// TIA Portal project "proyecto robot" (V15)

(* hardware
DEVICE "S7-1200 station_1"  S7-1200 Station
   slot 0: "Rack_0"  S7-1200 Rack  Rack  V1.0
   slot 1: "PLC_DERECHA"  CPU 1214C AC/DC/Rly  6ES7 214-1BG31-0XB0  V3.0
   slot 2: "AI 4x13BIT/AQ 2x14BIT_1"  6ES7 234-4HE32-0XB0  V2.0
DEVICE "S7-1200 station_2"  S7-1200 Station
   slot 0: "Rack_0"  S7-1200 Rack  Rack  V1.0
   slot 1: "PLC_IZQUIERDA"  CPU 1214C AC/DC/Rly  6ES7 214-1BG31-0XB0  V3.0
DEVICE "PC-System_1"  SIMATIC PC station
   slot 0: "Estación PC SIMATIC"  Rail  SIMATIC PC-Station  V1.0
      slot 125: "Stationmanager"  Station_Manager  V6.0.4
   slot 1: "HMI_RT_1"  WinCC RT Advanced  6AV2 104-0xxxx-xxxx  15.0.0.0
      slot 33792: "Interfaz host"  Host interface
   slot 2: "IE general_1"  IE General  IE_CP  V8.2.0
*)

// ===== PLC "PLC_DERECHA"  CPU 1214C AC/DC/Rly =====

VAR_GLOBAL   // PLC tag table "Tabla de variables estándar"
   "Clock_Byte" AT %MB1 : Byte;
   "Clock_10Hz" AT %M1.0 : Bool;
   "Clock_5Hz" AT %M1.1 : Bool;
   "Clock_2.5Hz" AT %M1.2 : Bool;
   "Clock_2Hz" AT %M1.3 : Bool;
   "Clock_1.25Hz" AT %M1.4 : Bool;
   "Clock_1Hz" AT %M1.5 : Bool;
   "Clock_0.625Hz" AT %M1.6 : Bool;
   "Clock_0.5Hz" AT %M1.7 : Bool;
   "Datos recibidos" AT %MW10 : Word;
   "Valor normalizado ultrasonidos" AT %MD50 : Real;
   "Distancia" AT %MD54 : Real;
   "Valor frecuencia cinta rueda" AT %MD58 : Real;
   "Valor normalizado frecuencia rueda" AT %MD62 : Real;
   "Normalizar frecuencia cinta chasis" AT %MD66 : Real;
   "Inicialización" AT %M12.0 : Bool;
   "marca cinta rueda" AT %M100.5 : Bool;
   "marca cilindro" AT %M100.6 : Bool;
   "Rueda en posición robot" AT %M11.1 : Bool;
   "Marca cinta chasis" AT %M100.4 : Bool;
   "Tag_4" AT %M100.7 : Bool;
   "Frecuencia cinta chasis" AT %MD70 : Real;
   "DISTANCIA HMI(1)" AT %MW200 : Int;
   "Cinta Lento" AT %MD204 : Real;
   "cinta nominal" AT %MD208 : Real;
   "HMI DISTANCIA" AT %MW1000 : Int;
   "Tag_1" AT %MD1000 : DWord;
   "Tag_2" AT %MD1200 : Real;
   "Tag_3" AT %MW500 : Word;
   "Tag_5" AT %MD500 : DInt;
   "Tag_6" AT %MD5005 : Real;
   "Tag_7" AT %MD504 : Real;
END_VAR

VAR_GLOBAL   // PLC tag table "Tabla de variables_1"
   "Error de comunicación" AT %M2.0 : Bool;
   "Marcha" AT %M10.0 : Bool;
   "Paro" AT %M10.1 : Bool;
   "Seta Emergencia" AT %M10.2 : Bool;
   "Fallo robot" AT %M10.3 : Bool;
   "jn rueda cilindro" AT %M10.4 : Bool;
   "jn fallo persona" AT %M10.5 : Bool;
   "jn cinta lento" AT %M10.6 : Bool;
   "guardamotor chasis" AT %M10.7 : Bool;
   "guardamotor rueda" AT %M11.0 : Bool;
   "Ultrasonidos" AT %IW96 : Word;
   "Variador cinta rueda" AT %QW96 : Word;
   "Variador cinta chasis" AT %QW98 : Word;
   "Motor cinta rueda" AT %Q0.0 : Bool;
   "Motor cinta chasis" AT %Q0.1 : Bool;
   "Cilindro" AT %Q0.2 : Bool;
   "Señal de fallo" AT %Q0.3 : Bool;
END_VAR

VAR_GLOBAL   // PLC tag table "HMI"
   "Seta emergencia HMI" AT %M20.0 : Bool;
   "Marcha HMI" AT %M20.1 : Bool;
   "Paro HMI" AT %M20.2 : Bool;
   "Marcha cinta chasis HMI" AT %M20.3 : Bool;
   "Paro cinta chasis HMI" AT %M20.4 : Bool;
   "Marcha cinta rueda HMI" AT %M20.5 : Bool;
   "Paro cinta rueda HMI" AT %M20.6 : Bool;
   "Control cilindro HMI" AT %M20.7 : Bool;
   "Luz marcha HMI" AT %M21.0 : Bool;
   "Luz paro HMI" AT %M21.1 : Bool;
   "Luz cinta chasis" AT %M21.2 : Bool;
   "Luz cinta rueda" AT %M21.3 : Bool;
   "Luz rueda en cinta" AT %M21.4 : Bool;
   "Luz cilindro fuera" AT %M21.5 : Bool;
   "Contador de tiempo" AT %MD300 : Time;
   "Tiempo" AT %MW202 : Word;
   "Luz seta emergencia" AT %M21.6 : Bool;
   "Luz fallo persona" AT %M21.7 : Bool;
   "Luz fallo robot" AT %M22.0 : Bool;
   "Luz guardamotor chasis" AT %M22.1 : Bool;
   "Luz guardamotor rueda" AT %M22.2 : Bool;
END_VAR

DATA_BLOCK "Guarda errores"   // DB3
{ S7_Optimized_Access := 'TRUE' }
VERSION : 0.1
   VAR
      "Seta emergencia" : DTL;
      "Fallo robot" : DTL;
      "Fallo persona" : DTL;
      "Guardamotor chasis" : DTL;
      "Guardamotor rueda" : DTL;
      "Retorno emergencia" : Int;
      "Retorno robot" : Int;
      "Retorno persona" : Int;
      "Retorno Guardamotor chasis" : Int;
      "Retorno guardamotor rueda" : Int;
   END_VAR
BEGIN
END_DATA_BLOCK

DATA_BLOCK "Velocidades"   // DB5
{ S7_Optimized_Access := 'TRUE' }
VERSION : 0.1
   VAR
      "Velocidad Lento" : Real := 10.5;
      "Velocidad Nominal" : Real := 40.0;
      "Velocidad cinta chasis" : Real := 5.0;
   END_VAR
BEGIN
END_DATA_BLOCK

// folder: System blocks/Program resources

DATA_BLOCK "PLC_DERECHA_Receive_DB"   // DB1
{ S7_Optimized_Access := 'TRUE' }
AUTHOR : SIMATIC
FAMILY : MC7Plus
NAME : TCON_Prm
VERSION : 1.0
// stored: InstanceOfName TCON_Param
"TCON_Param"
BEGIN
   ID := 1;
   REM_TSAP_ID_LEN := 0;
   LOCAL_TSAP_ID[1] := B#16#07;
   LOCAL_TSAP_ID[2] := B#16#D0;
   LOCAL_TSAP_ID_LEN := 2;
   ACTIVE_EST := false;
   REM_STADDR[1] := 172;
   REM_STADDR[2] := 26;
   REM_STADDR[3] := 20;
   REM_STADDR[4] := 50;
END_DATA_BLOCK

DATA_BLOCK "IEC_Timer_0_DB"   // DB4
{ S7_Optimized_Access := 'TRUE' }
AUTHOR : Simatic
FAMILY : IEC
NAME : IEC_TMR
VERSION : 1.0
// stored: InstanceOfName IEC_TIMER
"IEC_TIMER"
BEGIN
END_DATA_BLOCK

// folder: (top level)

FUNCTION "Cinta rueda" : Void   // FC1, LAD
{ S7_Optimized_Access := 'TRUE' }
VERSION : 0.1
   VAR_INPUT
      "Jetson Nano velocidad" : Bool;
      "Jetson Nano Rueda posición" : Bool;
      "Seta Emergencia" : Bool;
      "Fallo persona" : Bool;
      "Fallo robot" : Bool;
      Marcha : Bool;
      "Rueda abajo rampa" : Bool;
      Paro : Bool;
      "guardamotor chasis" : Bool;
      "guardamotor rueda" : Bool;
      Ultrasonidos : Real;
   END_VAR
   VAR_OUTPUT
      "Frecuencia cinta" : Int;
      "Activar cinta" : Bool;
   END_VAR
   VAR_IN_OUT
      Cilindro : Bool;
   END_VAR
BEGIN

REGION Network 1
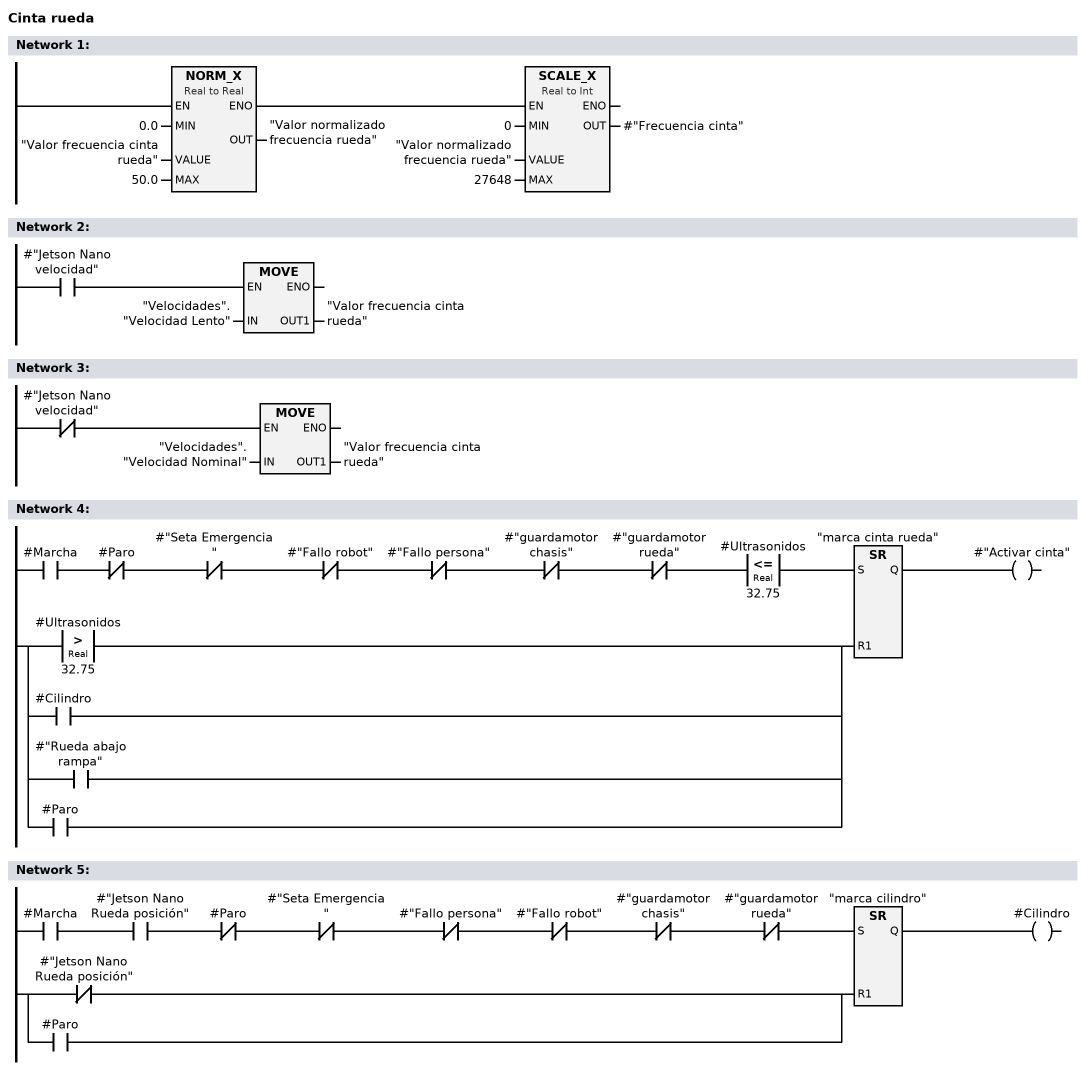
   RUNG wire#powerrail
      { S7_Templates := "[SrcType := Real, DestType := Real]"; S7_GenerateENO := "TRUE" } Normalize(min := 0.0, value := "Valor frecuencia cinta rueda", max := 50.0, out => "Valor normalizado frecuencia rueda")
      { S7_Templates := "[SrcType := Real, DestType := Int]"; S7_GenerateENO := "TRUE" } Scale(min := 0, value := "Valor normalizado frecuencia rueda", max := 27648, out => #"Frecuencia cinta")
   END_RUNG
   // the same network as SCL:
   // ENO of a box is taken as its EN; it also drops when the box reports an error
   "Valor normalizado frecuencia rueda" := NORM_X(MIN := 0.0, VALUE := "Valor frecuencia cinta rueda", MAX := 50.0);
   #"Frecuencia cinta" := SCALE_X(MIN := 0, VALUE := "Valor normalizado frecuencia rueda", MAX := 27648);
END_REGION

REGION Network 2
   RUNG wire#powerrail
      Contact( #"Jetson Nano velocidad" )
      { S7_GenerateENO := "TRUE" } Move(in := "Velocidades"."Velocidad Lento", out1 => "Valor frecuencia cinta rueda")
   END_RUNG
   // the same network as SCL:
   IF #"Jetson Nano velocidad" THEN
       "Valor frecuencia cinta rueda" := "Velocidades"."Velocidad Lento";
   END_IF;
END_REGION

REGION Network 3
   RUNG wire#powerrail
      I_Contact( #"Jetson Nano velocidad" )
      { S7_GenerateENO := "TRUE" } Move(in := "Velocidades"."Velocidad Nominal", out1 => "Valor frecuencia cinta rueda")
   END_RUNG
   // the same network as SCL:
   IF NOT #"Jetson Nano velocidad" THEN
       "Valor frecuencia cinta rueda" := "Velocidades"."Velocidad Nominal";
   END_IF;
END_REGION

REGION Network 4
   RUNG wire#powerrail
      Contact( #Marcha )
      I_Contact( #Paro )
      I_Contact( #"Seta Emergencia" )
      I_Contact( #"Fallo robot" )
      I_Contact( #"Fallo persona" )
      I_Contact( #"guardamotor chasis" )
      I_Contact( #"guardamotor rueda" )
      { S7_Templates := "SrcType := Real" } LE_Contact(in1 := #Ultrasonidos, in2 := 32.75)
      S_SR(operand := "marca cinta rueda", r1 := wire#w1)
      Coil( #"Activar cinta" )
   END_RUNG
   RUNG wire#powerrail
      { S7_Templates := "SrcType := Real" } GT_Contact(in1 := #Ultrasonidos, in2 := 32.75)
   END_RUNG wire#w1
   RUNG wire#powerrail
      Contact( #Cilindro )
   END_RUNG wire#w1
   RUNG wire#powerrail
      Contact( #"Rueda abajo rampa" )
   END_RUNG wire#w1
   RUNG wire#powerrail
      Contact( #Paro )
   END_RUNG wire#w1
   // the same network as SCL:
   IF #Marcha AND NOT #Paro AND NOT #"Seta Emergencia" AND NOT #"Fallo robot" AND NOT #"Fallo persona" AND NOT #"guardamotor chasis" AND NOT #"guardamotor rueda" AND (#Ultrasonidos <= 32.75) THEN
       "marca cinta rueda" := TRUE;   // SR flip-flop
   END_IF;
   IF (#Ultrasonidos > 32.75) OR #Cilindro OR #"Rueda abajo rampa" OR #Paro THEN
       "marca cinta rueda" := FALSE;
   END_IF;
   #"Activar cinta" := "marca cinta rueda";
END_REGION

REGION Network 5
   RUNG wire#powerrail
      Contact( #Marcha )
      Contact( #"Jetson Nano Rueda posición" )
      I_Contact( #Paro )
      I_Contact( #"Seta Emergencia" )
      I_Contact( #"Fallo persona" )
      I_Contact( #"Fallo robot" )
      I_Contact( #"guardamotor chasis" )
      I_Contact( #"guardamotor rueda" )
      S_SR(operand := "marca cilindro", r1 := wire#w1)
      Coil( #Cilindro )
   END_RUNG
   RUNG wire#powerrail
      I_Contact( #"Jetson Nano Rueda posición" )
   END_RUNG wire#w1
   RUNG wire#powerrail
      Contact( #Paro )
   END_RUNG wire#w1
   // the same network as SCL:
   IF #Marcha AND #"Jetson Nano Rueda posición" AND NOT #Paro AND NOT #"Seta Emergencia" AND NOT #"Fallo persona" AND NOT #"Fallo robot" AND NOT #"guardamotor chasis" AND NOT #"guardamotor rueda" THEN
       "marca cilindro" := TRUE;   // SR flip-flop
   END_IF;
   IF NOT #"Jetson Nano Rueda posición" OR #Paro THEN "marca cilindro" := FALSE; END_IF;
   #Cilindro := "marca cilindro";
END_REGION
END_FUNCTION

FUNCTION "Cinta chasis" : Void   // FC2, LAD
{ S7_Optimized_Access := 'TRUE' }
VERSION : 0.1
   VAR_INPUT
      Distancia : Real;
      Marcha : Bool;
      Paro : Bool;
      Emergencia : Bool;
      "Fallo persona" : Bool;
      "guardamotor chasis" : Bool;
      "guardamotor rueda" : Bool;
      "Fallo robot" : Bool;
   END_VAR
   VAR_OUTPUT
      "Activar cinta" : Bool;
      "Velocidad cinta" : Int;
   END_VAR
BEGIN

REGION Network 1
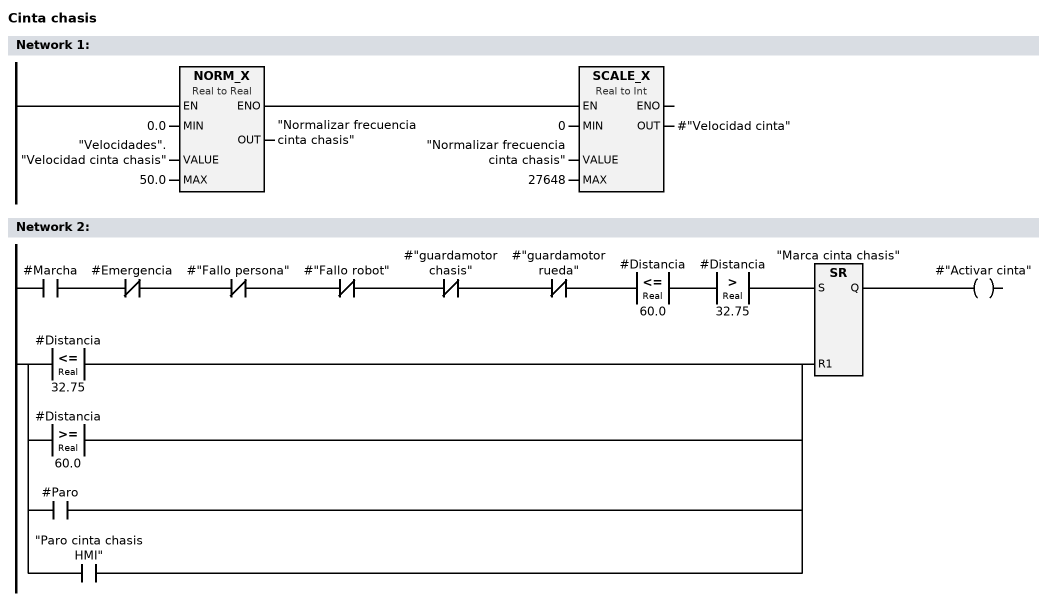
   RUNG wire#powerrail
      { S7_Templates := "[SrcType := Real, DestType := Real]"; S7_GenerateENO := "TRUE" } Normalize(min := 0.0, value := "Velocidades"."Velocidad cinta chasis", max := 50.0, out => "Normalizar frecuencia cinta chasis")
      { S7_Templates := "[SrcType := Real, DestType := Int]"; S7_GenerateENO := "TRUE" } Scale(min := 0, value := "Normalizar frecuencia cinta chasis", max := 27648, out => #"Velocidad cinta")
   END_RUNG
   // the same network as SCL:
   // ENO of a box is taken as its EN; it also drops when the box reports an error
   "Normalizar frecuencia cinta chasis" := NORM_X(MIN := 0.0, VALUE := "Velocidades"."Velocidad cinta chasis", MAX := 50.0);
   #"Velocidad cinta" := SCALE_X(MIN := 0, VALUE := "Normalizar frecuencia cinta chasis", MAX := 27648);
END_REGION

REGION Network 2
   RUNG wire#powerrail
      Contact( #Marcha )
      I_Contact( #Emergencia )
      I_Contact( #"Fallo persona" )
      I_Contact( #"Fallo robot" )
      I_Contact( #"guardamotor chasis" )
      I_Contact( #"guardamotor rueda" )
      { S7_Templates := "SrcType := Real" } LE_Contact(in1 := #Distancia, in2 := 60.0)
      { S7_Templates := "SrcType := Real" } GT_Contact(in1 := #Distancia, in2 := 32.75)
      S_SR(operand := "Marca cinta chasis", r1 := wire#w1)
      Coil( #"Activar cinta" )
   END_RUNG
   RUNG wire#powerrail
      { S7_Templates := "SrcType := Real" } LE_Contact(in1 := #Distancia, in2 := 32.75)
   END_RUNG wire#w1
   RUNG wire#powerrail
      { S7_Templates := "SrcType := Real" } GE_Contact(in1 := #Distancia, in2 := 60.0)
   END_RUNG wire#w1
   RUNG wire#powerrail
      Contact( #Paro )
   END_RUNG wire#w1
   RUNG wire#powerrail
      Contact( "Paro cinta chasis HMI" )
   END_RUNG wire#w1
   // the same network as SCL:
   IF #Marcha AND NOT #Emergencia AND NOT #"Fallo persona" AND NOT #"Fallo robot" AND NOT #"guardamotor chasis" AND NOT #"guardamotor rueda" AND (#Distancia <= 60.0) AND (#Distancia > 32.75) THEN
       "Marca cinta chasis" := TRUE;   // SR flip-flop
   END_IF;
   IF (#Distancia <= 32.75) OR (#Distancia >= 60.0) OR #Paro OR "Paro cinta chasis HMI" THEN
       "Marca cinta chasis" := FALSE;
   END_IF;
   #"Activar cinta" := "Marca cinta chasis";
END_REGION
END_FUNCTION

FUNCTION "Emergencias" : Void   // FC3, LAD
TITLE = EMERGENCIAS
{ S7_Optimized_Access := 'TRUE' }
VERSION : 0.1
   VAR_INPUT
      Emergencia : Bool;
      "Fallo Persona" : Bool;
      "Fallo Robot" : Bool;
      "Guardamotor chasis" : Bool;
      "Guardamotor rueda" : Bool;
   END_VAR
   VAR_OUTPUT
      "Salida de Fallo" : Bool;
      "Cinta Chasis" : Bool;
      "Cinta rueda" : Bool;
      Cilindro : Bool;
   END_VAR
BEGIN

REGION Network 1: DESACTIVAR CINTA CHASIS
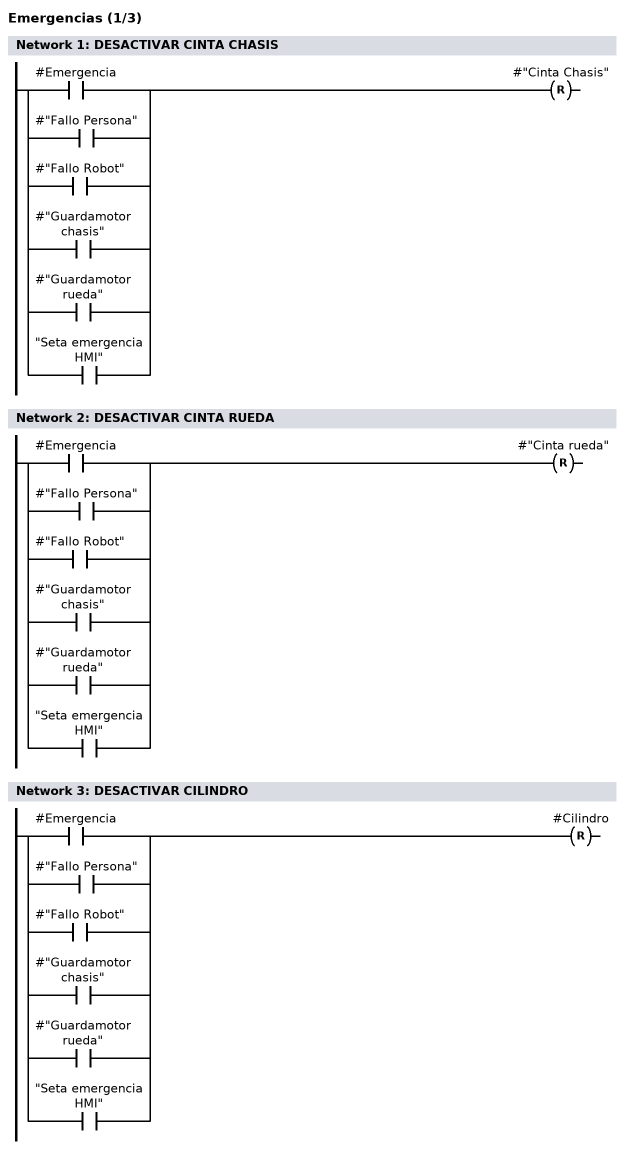
   RUNG wire#powerrail
      Contact( #Emergencia )
      wire#w1
      R_Coil( #"Cinta Chasis" )
   END_RUNG
   RUNG wire#powerrail
      Contact( #"Fallo Persona" )
   END_RUNG wire#w1
   RUNG wire#powerrail
      Contact( #"Fallo Robot" )
   END_RUNG wire#w1
   RUNG wire#powerrail
      Contact( #"Guardamotor chasis" )
   END_RUNG wire#w1
   RUNG wire#powerrail
      Contact( #"Guardamotor rueda" )
   END_RUNG wire#w1
   RUNG wire#powerrail
      Contact( "Seta emergencia HMI" )
   END_RUNG wire#w1
   // the same network as SCL:
   IF #Emergencia OR #"Fallo Persona" OR #"Fallo Robot" OR #"Guardamotor chasis" OR #"Guardamotor rueda" OR "Seta emergencia HMI" THEN
       #"Cinta Chasis" := FALSE;
   END_IF;
END_REGION

REGION Network 2: DESACTIVAR CINTA RUEDA
   RUNG wire#powerrail
      Contact( #Emergencia )
      wire#w1
      R_Coil( #"Cinta rueda" )
   END_RUNG
   RUNG wire#powerrail
      Contact( #"Fallo Persona" )
   END_RUNG wire#w1
   RUNG wire#powerrail
      Contact( #"Fallo Robot" )
   END_RUNG wire#w1
   RUNG wire#powerrail
      Contact( #"Guardamotor chasis" )
   END_RUNG wire#w1
   RUNG wire#powerrail
      Contact( #"Guardamotor rueda" )
   END_RUNG wire#w1
   RUNG wire#powerrail
      Contact( "Seta emergencia HMI" )
   END_RUNG wire#w1
   // the same network as SCL:
   IF #Emergencia OR #"Fallo Persona" OR #"Fallo Robot" OR #"Guardamotor chasis" OR #"Guardamotor rueda" OR "Seta emergencia HMI" THEN
       #"Cinta rueda" := FALSE;
   END_IF;
END_REGION

REGION Network 3: DESACTIVAR CILINDRO
   RUNG wire#powerrail
      Contact( #Emergencia )
      wire#w1
      R_Coil( #Cilindro )
   END_RUNG
   RUNG wire#powerrail
      Contact( #"Fallo Persona" )
   END_RUNG wire#w1
   RUNG wire#powerrail
      Contact( #"Fallo Robot" )
   END_RUNG wire#w1
   RUNG wire#powerrail
      Contact( #"Guardamotor chasis" )
   END_RUNG wire#w1
   RUNG wire#powerrail
      Contact( #"Guardamotor rueda" )
   END_RUNG wire#w1
   RUNG wire#powerrail
      Contact( "Seta emergencia HMI" )
   END_RUNG wire#w1
   // the same network as SCL:
   IF #Emergencia OR #"Fallo Persona" OR #"Fallo Robot" OR #"Guardamotor chasis" OR #"Guardamotor rueda" OR "Seta emergencia HMI" THEN
       #Cilindro := FALSE;
   END_IF;
END_REGION

REGION Network 4: SALIDA FALLO
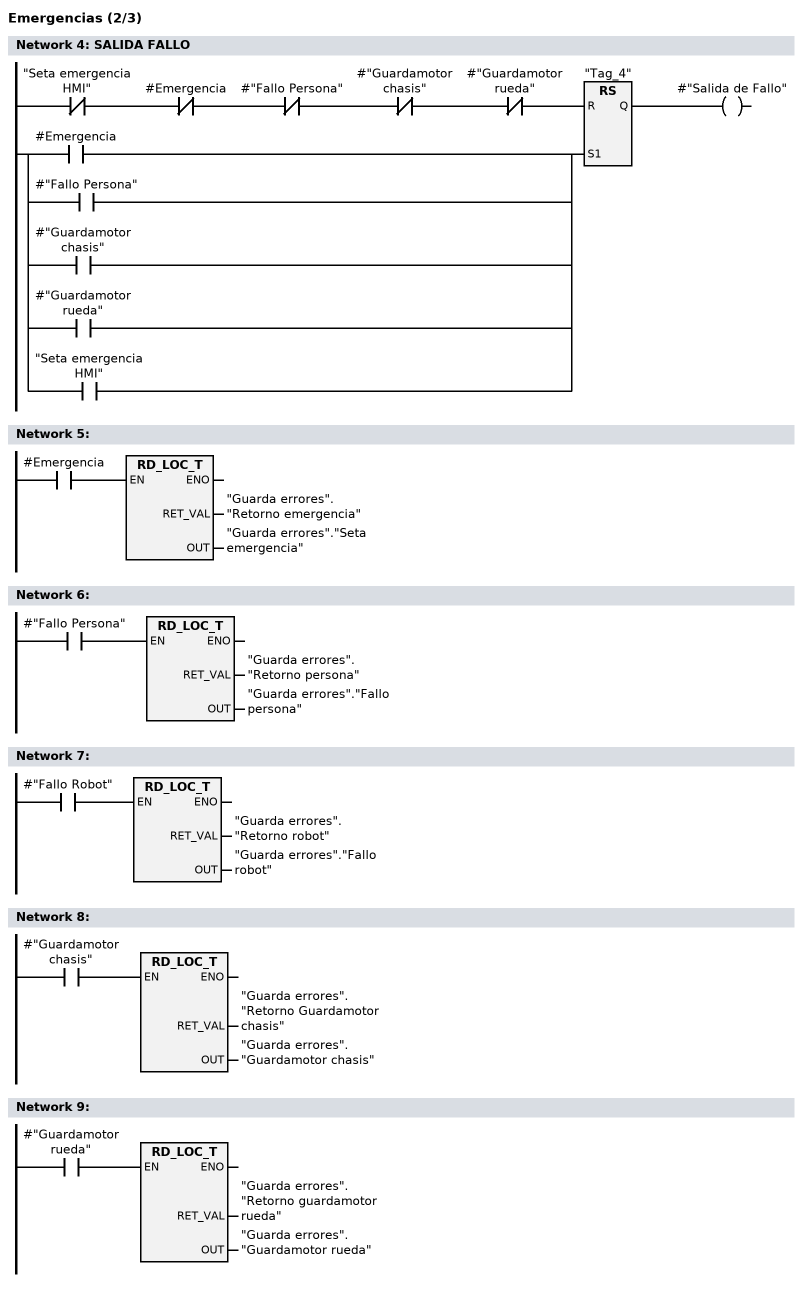
   RUNG wire#powerrail
      I_Contact( "Seta emergencia HMI" )
      I_Contact( #Emergencia )
      I_Contact( #"Fallo Persona" )
      I_Contact( #"Guardamotor chasis" )
      I_Contact( #"Guardamotor rueda" )
      S_RS(operand := "Tag_4", s1 := wire#w1)
      Coil( #"Salida de Fallo" )
   END_RUNG
   RUNG wire#powerrail
      Contact( #Emergencia )
   END_RUNG wire#w1
   RUNG wire#powerrail
      Contact( #"Fallo Persona" )
   END_RUNG wire#w1
   RUNG wire#powerrail
      Contact( #"Guardamotor chasis" )
   END_RUNG wire#w1
   RUNG wire#powerrail
      Contact( #"Guardamotor rueda" )
   END_RUNG wire#w1
   RUNG wire#powerrail
      Contact( "Seta emergencia HMI" )
   END_RUNG wire#w1
   // the same network as SCL:
   IF NOT "Seta emergencia HMI" AND NOT #Emergencia AND NOT #"Fallo Persona" AND NOT #"Guardamotor chasis" AND NOT #"Guardamotor rueda" THEN
       "Tag_4" := FALSE;   // RS flip-flop
   END_IF;
   IF #Emergencia OR #"Fallo Persona" OR #"Guardamotor chasis" OR #"Guardamotor rueda" OR "Seta emergencia HMI" THEN
       "Tag_4" := TRUE;
   END_IF;
   #"Salida de Fallo" := "Tag_4";
END_REGION

REGION Network 5
   IF #Emergencia THEN
       "Guarda errores"."Retorno emergencia" := RD_LOC_T(OUT => "Guarda errores"."Seta emergencia");
   END_IF;
END_REGION

REGION Network 6
   IF #"Fallo Persona" THEN
       "Guarda errores"."Retorno persona" := RD_LOC_T(OUT => "Guarda errores"."Fallo persona");
   END_IF;
END_REGION

REGION Network 7
   IF #"Fallo Robot" THEN
       "Guarda errores"."Retorno robot" := RD_LOC_T(OUT => "Guarda errores"."Fallo robot");
   END_IF;
END_REGION

REGION Network 8
   IF #"Guardamotor chasis" THEN
       "Guarda errores"."Retorno Guardamotor chasis" := RD_LOC_T(OUT => "Guarda errores"."Guardamotor chasis");
   END_IF;
END_REGION

REGION Network 9
   IF #"Guardamotor rueda" THEN
       "Guarda errores"."Retorno guardamotor rueda" := RD_LOC_T(OUT => "Guarda errores"."Guardamotor rueda");
   END_IF;
END_REGION

REGION Network 10
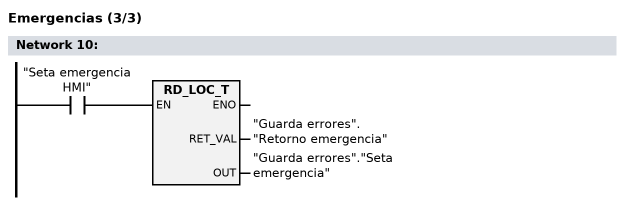
   IF "Seta emergencia HMI" THEN
       "Guarda errores"."Retorno emergencia" := RD_LOC_T(OUT => "Guarda errores"."Seta emergencia");
   END_IF;
END_REGION
END_FUNCTION

FUNCTION "HMI" : Void   // FC4, LAD
{ S7_Optimized_Access := 'TRUE' }
VERSION : 0.1
BEGIN

REGION Network 1
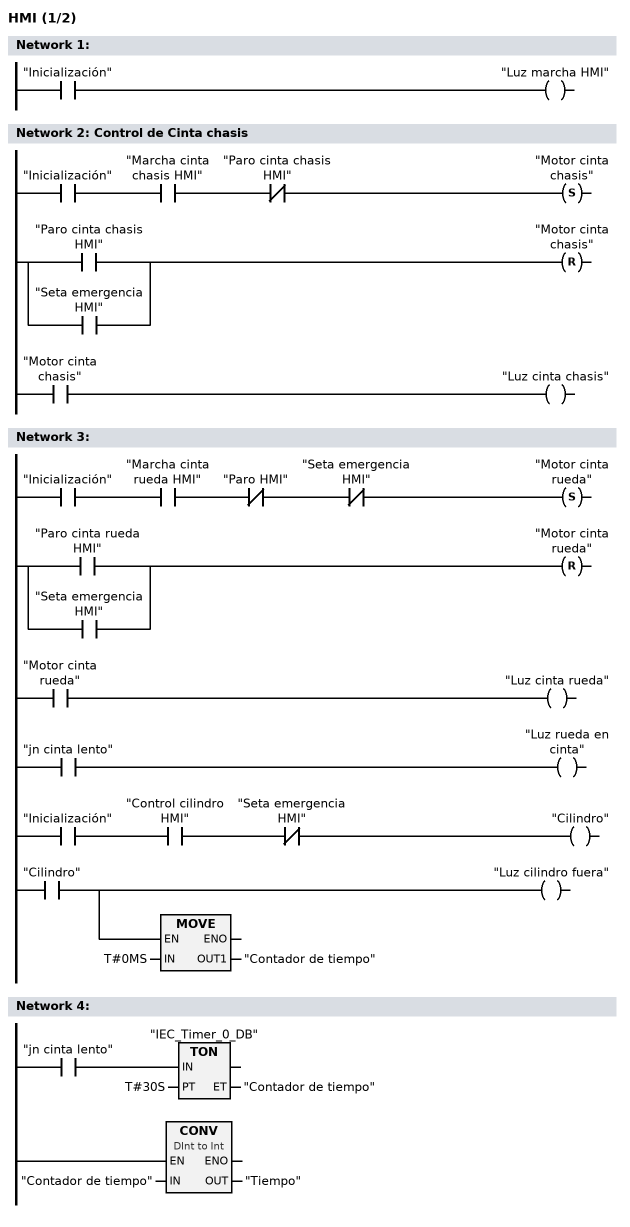
   RUNG wire#powerrail
      Contact( "Inicialización" )
      Coil( "Luz marcha HMI" )
   END_RUNG
   // the same network as SCL:
   "Luz marcha HMI" := "Inicialización";
END_REGION

REGION Network 2: Control de Cinta chasis
   RUNG wire#powerrail
      Contact( "Inicialización" )
      Contact( "Marcha cinta chasis HMI" )
      I_Contact( "Paro cinta chasis HMI" )
      S_Coil( "Motor cinta chasis" )
   END_RUNG
   RUNG wire#powerrail
      Contact( "Paro cinta chasis HMI" )
      wire#w1
      R_Coil( "Motor cinta chasis" )
   END_RUNG
   RUNG wire#powerrail
      Contact( "Seta emergencia HMI" )
   END_RUNG wire#w1
   RUNG wire#powerrail
      Contact( "Motor cinta chasis" )
      Coil( "Luz cinta chasis" )
   END_RUNG
   // the same network as SCL:
   IF "Inicialización" AND "Marcha cinta chasis HMI" AND NOT "Paro cinta chasis HMI" THEN
       "Motor cinta chasis" := TRUE;
   END_IF;
   IF "Paro cinta chasis HMI" OR "Seta emergencia HMI" THEN "Motor cinta chasis" := FALSE; END_IF;
   "Luz cinta chasis" := "Motor cinta chasis";
END_REGION

REGION Network 3
   RUNG wire#powerrail
      Contact( "Inicialización" )
      Contact( "Marcha cinta rueda HMI" )
      I_Contact( "Paro HMI" )
      I_Contact( "Seta emergencia HMI" )
      S_Coil( "Motor cinta rueda" )
   END_RUNG
   RUNG wire#powerrail
      Contact( "Paro cinta rueda HMI" )
      wire#w1
      R_Coil( "Motor cinta rueda" )
   END_RUNG
   RUNG wire#powerrail
      Contact( "Seta emergencia HMI" )
   END_RUNG wire#w1
   RUNG wire#powerrail
      Contact( "Motor cinta rueda" )
      Coil( "Luz cinta rueda" )
   END_RUNG
   RUNG wire#powerrail
      Contact( "jn cinta lento" )
      Coil( "Luz rueda en cinta" )
   END_RUNG
   RUNG wire#powerrail
      Contact( "Inicialización" )
      Contact( "Control cilindro HMI" )
      I_Contact( "Seta emergencia HMI" )
      Coil( "Cilindro" )
   END_RUNG
   RUNG wire#powerrail
      Contact( "Cilindro" )
      wire#w2
      Coil( "Luz cilindro fuera" )
   END_RUNG
   RUNG wire#w2
      { S7_GenerateENO := "TRUE" } Move(in := T#0MS, out1 => "Contador de tiempo")
   END_RUNG
   // the same network as SCL:
   IF "Inicialización" AND "Marcha cinta rueda HMI" AND NOT "Paro HMI" AND NOT "Seta emergencia HMI" THEN
       "Motor cinta rueda" := TRUE;
   END_IF;
   IF "Paro cinta rueda HMI" OR "Seta emergencia HMI" THEN "Motor cinta rueda" := FALSE; END_IF;
   "Luz cinta rueda" := "Motor cinta rueda";
   "Luz rueda en cinta" := "jn cinta lento";
   "Cilindro" := "Inicialización" AND "Control cilindro HMI" AND NOT "Seta emergencia HMI";
   "Luz cilindro fuera" := "Cilindro";
   IF "Cilindro" THEN "Contador de tiempo" := T#0MS; END_IF;
END_REGION

REGION Network 4
   "IEC_Timer_0_DB".TON(IN := "jn cinta lento", PT := T#30S, ET => "Contador de tiempo");
   "Tiempo" := DINT_TO_INT("Contador de tiempo");
END_REGION

REGION Network 6: LUCES DE EMERGENCIA
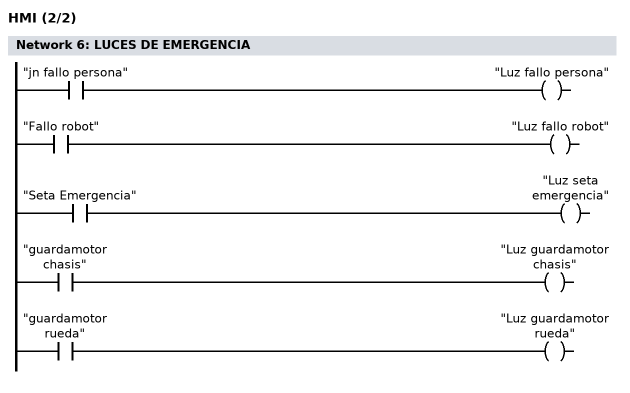
   RUNG wire#powerrail
      Contact( "jn fallo persona" )
      Coil( "Luz fallo persona" )
   END_RUNG
   RUNG wire#powerrail
      Contact( "Fallo robot" )
      Coil( "Luz fallo robot" )
   END_RUNG
   RUNG wire#powerrail
      Contact( "Seta Emergencia" )
      Coil( "Luz seta emergencia" )
   END_RUNG
   RUNG wire#powerrail
      Contact( "guardamotor chasis" )
      Coil( "Luz guardamotor chasis" )
   END_RUNG
   RUNG wire#powerrail
      Contact( "guardamotor rueda" )
      Coil( "Luz guardamotor rueda" )
   END_RUNG
   // the same network as SCL:
   "Luz fallo persona" := "jn fallo persona";
   "Luz fallo robot" := "Fallo robot";
   "Luz seta emergencia" := "Seta Emergencia";
   "Luz guardamotor chasis" := "guardamotor chasis";
   "Luz guardamotor rueda" := "guardamotor rueda";
END_REGION
END_FUNCTION

ORGANIZATION_BLOCK "Main"   // OB1, LAD, ProgramCycle
TITLE = "Main Program Sweep (Cycle)"
{ S7_Optimized_Access := 'TRUE' }
VERSION : 0.1
BEGIN

REGION Network 1
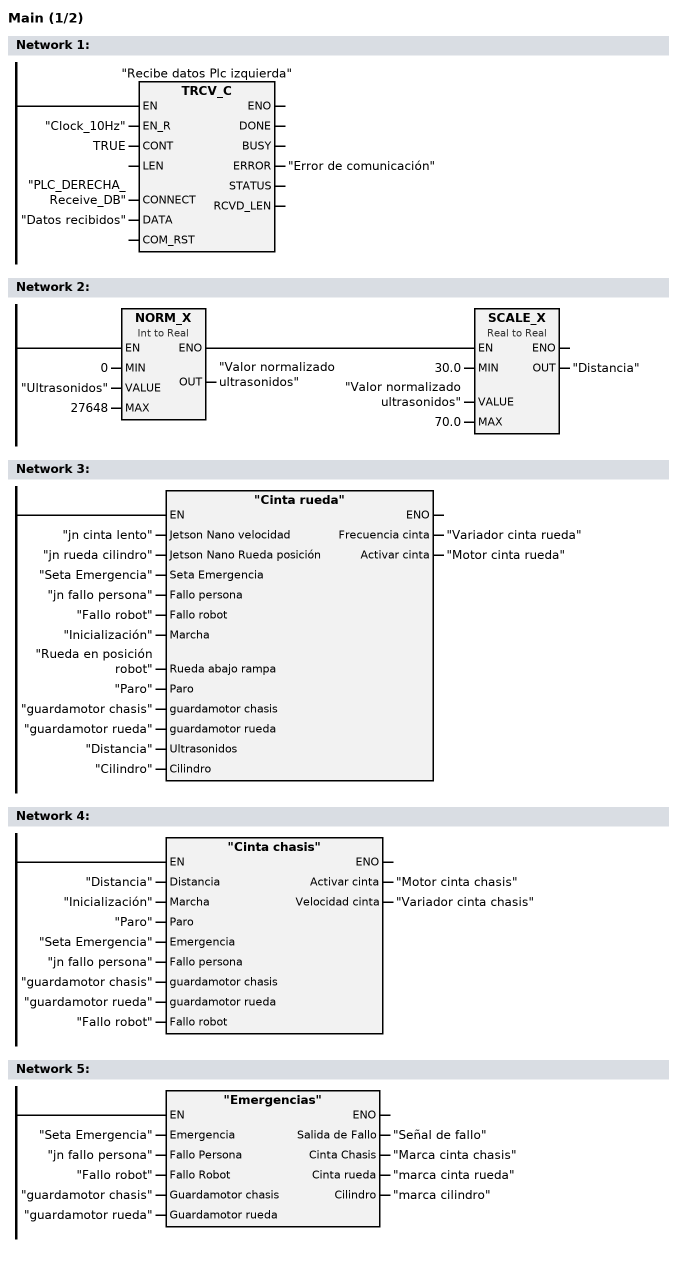
   "Recibe datos Plc izquierda"(EN_R := "Clock_10Hz",   // TRCV_C
                           CONT := TRUE,
                           CONNECT := "PLC_DERECHA_Receive_DB",
                           DATA := "Datos recibidos",
                           ERROR => "Error de comunicación");
END_REGION

REGION Network 2
   RUNG wire#powerrail
      { S7_Templates := "[SrcType := Int, DestType := Real]"; S7_GenerateENO := "TRUE" } Normalize(min := 0, value := "Ultrasonidos", max := 27648, out => "Valor normalizado ultrasonidos")
      { S7_Templates := "[SrcType := Real, DestType := Real]"; S7_GenerateENO := "TRUE" } Scale(min := 30.0, value := "Valor normalizado ultrasonidos", max := 70.0, out => "Distancia")
   END_RUNG
   // the same network as SCL:
   // ENO of a box is taken as its EN; it also drops when the box reports an error
   "Valor normalizado ultrasonidos" := NORM_X(MIN := 0, VALUE := "Ultrasonidos", MAX := 27648);
   "Distancia" := SCALE_X(MIN := 30.0, VALUE := "Valor normalizado ultrasonidos", MAX := 70.0);
END_REGION

REGION Network 3
   RUNG wire#powerrail
      "Cinta rueda"("Jetson Nano velocidad" := "jn cinta lento", "Jetson Nano Rueda posición" := "jn rueda cilindro", "Seta Emergencia" := "Seta Emergencia", "Fallo persona" := "jn fallo persona", "Fallo robot" := "Fallo robot", Marcha := "Inicialización", "Rueda abajo rampa" := "Rueda en posición robot", Paro := "Paro", "guardamotor chasis" := "guardamotor chasis", "guardamotor rueda" := "guardamotor rueda", Ultrasonidos := "Distancia", Cilindro := "Cilindro", "Frecuencia cinta" => "Variador cinta rueda", "Activar cinta" => "Motor cinta rueda")
   END_RUNG
   // the same network as SCL:
   "Cinta rueda"("Jetson Nano velocidad" := "jn cinta lento",
                 "Jetson Nano Rueda posición" := "jn rueda cilindro",
                 "Seta Emergencia" := "Seta Emergencia",
                 "Fallo persona" := "jn fallo persona",
                 "Fallo robot" := "Fallo robot",
                 Marcha := "Inicialización",
                 "Rueda abajo rampa" := "Rueda en posición robot",
                 Paro := "Paro",
                 "guardamotor chasis" := "guardamotor chasis",
                 "guardamotor rueda" := "guardamotor rueda",
                 Ultrasonidos := "Distancia",
                 Cilindro := "Cilindro",
                 "Frecuencia cinta" => "Variador cinta rueda",
                 "Activar cinta" => "Motor cinta rueda");
END_REGION

REGION Network 4
   RUNG wire#powerrail
      "Cinta chasis"(Distancia := "Distancia", Marcha := "Inicialización", Paro := "Paro", Emergencia := "Seta Emergencia", "Fallo persona" := "jn fallo persona", "guardamotor chasis" := "guardamotor chasis", "guardamotor rueda" := "guardamotor rueda", "Fallo robot" := "Fallo robot", "Activar cinta" => "Motor cinta chasis", "Velocidad cinta" => "Variador cinta chasis")
   END_RUNG
   // the same network as SCL:
   "Cinta chasis"(Distancia := "Distancia",
                  Marcha := "Inicialización",
                  Paro := "Paro",
                  Emergencia := "Seta Emergencia",
                  "Fallo persona" := "jn fallo persona",
                  "guardamotor chasis" := "guardamotor chasis",
                  "guardamotor rueda" := "guardamotor rueda",
                  "Fallo robot" := "Fallo robot",
                  "Activar cinta" => "Motor cinta chasis",
                  "Velocidad cinta" => "Variador cinta chasis");
END_REGION

REGION Network 5
   RUNG wire#powerrail
      "Emergencias"(Emergencia := "Seta Emergencia", "Fallo Persona" := "jn fallo persona", "Fallo Robot" := "Fallo robot", "Guardamotor chasis" := "guardamotor chasis", "Guardamotor rueda" := "guardamotor rueda", "Salida de Fallo" => "Señal de fallo", "Cinta Chasis" => "Marca cinta chasis", "Cinta rueda" => "marca cinta rueda", Cilindro => "marca cilindro")
   END_RUNG
   // the same network as SCL:
   "Emergencias"(Emergencia := "Seta Emergencia",
                 "Fallo Persona" := "jn fallo persona",
                 "Fallo Robot" := "Fallo robot",
                 "Guardamotor chasis" := "guardamotor chasis",
                 "Guardamotor rueda" := "guardamotor rueda",
                 "Salida de Fallo" => "Señal de fallo",
                 "Cinta Chasis" => "Marca cinta chasis",
                 "Cinta rueda" => "marca cinta rueda",
                 Cilindro => "marca cilindro");
END_REGION

REGION Network 6
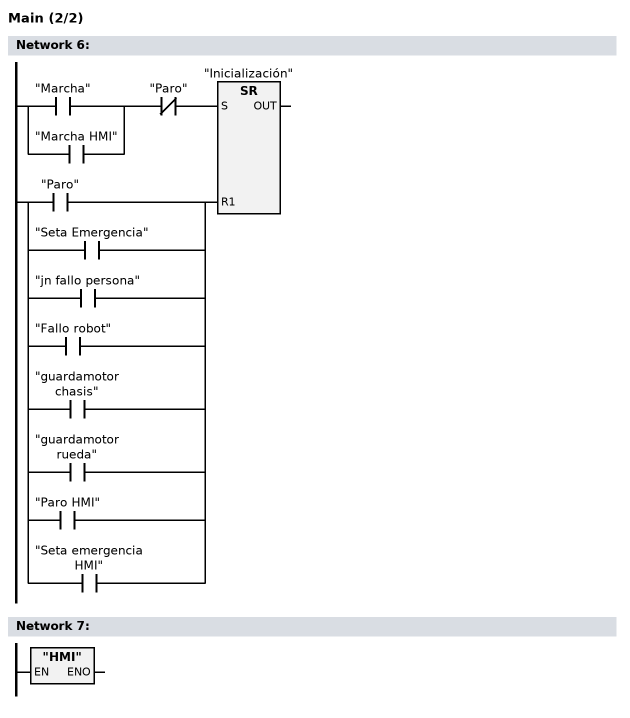
   RUNG wire#powerrail
      Contact( "Marcha" )
      wire#w1
      I_Contact( "Paro" )
      S_SR(operand := "Inicialización", r1 := wire#w2)
   END_RUNG
   RUNG wire#powerrail
      Contact( "Marcha HMI" )
   END_RUNG wire#w1
   RUNG wire#powerrail
      Contact( "Paro" )
   END_RUNG wire#w2
   RUNG wire#powerrail
      Contact( "Seta Emergencia" )
   END_RUNG wire#w2
   RUNG wire#powerrail
      Contact( "jn fallo persona" )
   END_RUNG wire#w2
   RUNG wire#powerrail
      Contact( "Fallo robot" )
   END_RUNG wire#w2
   RUNG wire#powerrail
      Contact( "guardamotor chasis" )
   END_RUNG wire#w2
   RUNG wire#powerrail
      Contact( "guardamotor rueda" )
   END_RUNG wire#w2
   RUNG wire#powerrail
      Contact( "Paro HMI" )
   END_RUNG wire#w2
   RUNG wire#powerrail
      Contact( "Seta emergencia HMI" )
   END_RUNG wire#w2
   // the same network as SCL:
   IF ("Marcha" OR "Marcha HMI") AND NOT "Paro" THEN
       "Inicialización" := TRUE;   // SR flip-flop
   END_IF;
   IF "Paro" OR "Seta Emergencia" OR "jn fallo persona" OR "Fallo robot" OR "guardamotor chasis" OR "guardamotor rueda" OR "Paro HMI" OR "Seta emergencia HMI" THEN
       "Inicialización" := FALSE;
   END_IF;
END_REGION

REGION Network 7
   RUNG wire#powerrail
      "HMI"()
   END_RUNG
   // the same network as SCL:
   "HMI"();
END_REGION
END_ORGANIZATION_BLOCK

// ===== PLC "PLC_IZQUIERDA"  CPU 1214C AC/DC/Rly =====

VAR_GLOBAL   // PLC tag table "Tabla de variables estándar"
   "Clock_Byte" AT %MB1 : Byte;
   "Clock_10Hz" AT %M1.0 : Bool;
   "Clock_5Hz" AT %M1.1 : Bool;
   "Clock_2.5Hz" AT %M1.2 : Bool;
   "Clock_2Hz" AT %M1.3 : Bool;
   "Clock_1.25Hz" AT %M1.4 : Bool;
   "Clock_1Hz" AT %M1.5 : Bool;
   "Clock_0.625Hz" AT %M1.6 : Bool;
   "Clock_0.5Hz" AT %M1.7 : Bool;
   "Datos a enviar" AT %IW0 : Word;
   "Tag_1" AT %M0.0 : Bool;
   "Tag_2" AT %M10.0 : Bool;
END_VAR

VAR_GLOBAL   // PLC tag table "Tabla de variables_1"
   "marcha" AT %I0.0 : Bool;
   "paro" AT %I0.1 : Bool;
   "Seta emergencia" AT %I0.2 : Bool;
   "fallo robot" AT %I0.3 : Bool;
   "jn rueda cilindro" AT %I0.4 : Bool;
   "jn fallo persona" AT %I0.5 : Bool;
   "jn cinta lento" AT %I0.6 : Bool;
   "guardamotor chasis" AT %I0.7 : Bool;
   "guardamotor rueda" AT %I1.0 : Bool;
END_VAR

// folder: System blocks/Program resources

DATA_BLOCK "PLC_IZQUIERDA_Send_DB"   // DB2
{ S7_Optimized_Access := 'TRUE' }
AUTHOR : SIMATIC
FAMILY : MC7Plus
NAME : TCON_Prm
VERSION : 1.0
// stored: InstanceOfName TCON_Param
"TCON_Param"
BEGIN
   ID := 1;
   REM_TSAP_ID[1] := B#16#07;
   REM_TSAP_ID[2] := B#16#D0;
   REM_STADDR[1] := 172;
   REM_STADDR[2] := 26;
   REM_STADDR[3] := 20;
   REM_STADDR[4] := 51;
END_DATA_BLOCK

// folder: (top level)

ORGANIZATION_BLOCK "Main"   // OB1, LAD, ProgramCycle
TITLE = "Main Program Sweep (Cycle)"
{ S7_Optimized_Access := 'TRUE' }
VERSION : 0.1
BEGIN

REGION Network 1
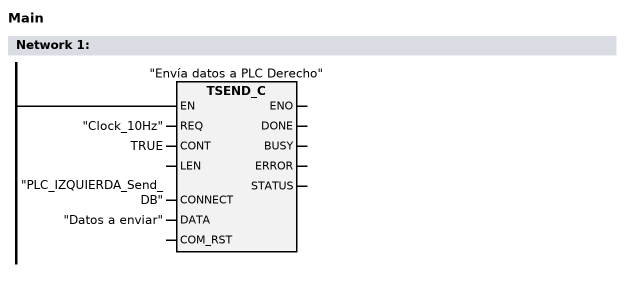
   "Envía datos a PLC Derecho"(REQ := "Clock_10Hz",   // TSEND_C
                           CONT := TRUE,
                           CONNECT := "PLC_IZQUIERDA_Send_DB",
                           DATA := "Datos a enviar");
END_REGION
END_ORGANIZATION_BLOCK

(* ===== HMI "HMI_RT_1" =====
system functions are stored by id; their names below are inferred from use
connection "HMI_Conexión_1": ETHERNET, S7_1200_OMS

HMI tags "Tabla de variables estándar"
   "Nombre_Usuario" : WString[10], internal
   "Es necesario autentificar" : Int, internal
   "Marcha cinta chasis HMI" : Bool = PLC "Marcha cinta chasis HMI" AT %M20.3, 1 s
   "Paro cinta chasis HMI" : Bool = PLC "Paro cinta chasis HMI" AT %M20.4, 1 s
   "Luz cinta chasis" : Bool = PLC "Luz cinta chasis" AT %M21.2, 1 s
   "Marcha cinta rueda HMI" : Bool = PLC "Marcha cinta rueda HMI" AT %M20.5, 1 s
   "Paro cinta rueda HMI" : Bool = PLC "Paro cinta rueda HMI" AT %M20.6, 1 s
   "Luz cinta rueda" : Bool = PLC "Luz cinta rueda" AT %M21.3, 1 s
   "Luz rueda en cinta" : Bool = PLC "Luz rueda en cinta" AT %M21.4, 1 s
   "Luz cilindro fuera" : Bool = PLC "Luz cilindro fuera" AT %M21.5, 1 s
   "Control cilindro HMI" : Bool = PLC "Control cilindro HMI" AT %M20.7, 1 s
   "Marcha HMI" : Bool = PLC "Marcha HMI" AT %M20.1, 1 s
   "Paro HMI" : Bool = PLC "Paro HMI" AT %M20.2, 1 s
   "Seta emergencia HMI" : Bool = PLC "Seta emergencia HMI" AT %M20.0, 1 s
   "Valor frecuencia cinta rueda" : Real = PLC "Valor frecuencia cinta rueda" AT %MD58, 1 s
   "Frecuencia cinta chasis" : Real = PLC "Frecuencia cinta chasis" AT %MD70, 1 s
   "Distancia" : Real = PLC Distancia AT %MD54, 1 s
   "Valor normalizado frecuencia rueda" : Real = PLC "Valor normalizado frecuencia rueda" AT %MD62, 1 s
   "Luz marcha HMI" : Bool = PLC "Luz marcha HMI" AT %M21.0, 1 s
   "DISTANCIA HMI(1)" : Int = PLC "DISTANCIA HMI(1)" AT %MW200, 1 s
   "marca cilindro" : Bool = PLC "marca cilindro" AT %M100.6, 1 s
   "Contador de tiempo" : Time = PLC "Contador de tiempo" AT %MD300, 1 s
   "jn cinta lento" : Bool = PLC "jn cinta lento" AT %M10.6, 1 s
   "cinta nominal" : Real = PLC "cinta nominal" AT %MD208, 1 s
   "Cinta Lento" : Real = PLC "Cinta Lento" AT %MD204, 1 s
   "Tiempo" : Word = PLC Tiempo AT %MW202, 1 s
   "Ultrasonidos" : Word = PLC Ultrasonidos AT %IW96, 1 s
   "HMI DISTANCIA" : Int = PLC "HMI DISTANCIA" AT %MW1000, 1 s
   "Tag_1" : DWord = PLC Tag_1 AT %MD1000, 1 s
   "Tag_3" : Word = PLC Tag_3 AT %MW500, 1 s
   "Tag_7" : Real = PLC Tag_7 AT %MD504, 1 s
   "Guarda errores_Seta emergencia" : DTL = PLC "Guarda errores"."Seta emergencia", 1 s
   "Guarda errores_Fallo persona" : DTL = PLC "Guarda errores"."Fallo persona", 1 s
   "Guarda errores_Fallo robot" : DTL = PLC "Guarda errores"."Fallo robot", 1 s
   "Guarda errores_Guardamotor chasis" : DTL = PLC "Guarda errores"."Guardamotor chasis", 1 s
   "Guarda errores_Guardamotor rueda" : DTL = PLC "Guarda errores"."Guardamotor rueda", 1 s
   "Luz seta emergencia" : Bool = PLC "Luz seta emergencia" AT %M21.6, 1 s
   "Luz fallo persona" : Bool = PLC "Luz fallo persona" AT %M21.7, 1 s
   "Luz fallo robot" : Bool = PLC "Luz fallo robot" AT %M22.0, 1 s
   "Luz guardamotor chasis" : Bool = PLC "Luz guardamotor chasis" AT %M22.1, 1 s
   "Luz guardamotor rueda" : Bool = PLC "Luz guardamotor rueda" AT %M22.2, 1 s
   "Velocidades_Velocidad cinta chasis" : Real = PLC Velocidades."Velocidad cinta chasis", 1 s
   "Velocidades_Velocidad Nominal" : Real = PLC Velocidades."Velocidad Nominal", 1 s
   "Velocidades_Velocidad Lento" : Real = PLC Velocidades."Velocidad Lento", 1 s

graphic list "Lista de gráficos_1": 0..1 'gratis-png-boton-de-flecha-flecha-de-retroceso-thumbnail'

Template "Plantilla_1" 800x600
   Button "SB_ExitRuntime_48x48" at 910,676 size 48x48; TextOff 'Text'; PictureOff "SB_ExitRuntime_48x48_256c"
      on Click: StopRuntime(0)
   GraphicView "Plantilla_Visor de gráficos_1" at 0,0 size 261x70; Picture "Logo-Manuel-Lora-Tamayo-2"
   TextField "Plantilla_Campo de texto_1" at 271,24 size 358x22; Text 'PROCESO DE FABRICACIÓN DE UN AUTOMÓVIL'
   DateTimeField "Plantilla_Campo de fecha y hora_1" at 634,1 size 166x69
   DateTimeField "Plantilla_Campo de fecha y hora_2" at 695,35 size 78x34
   TextField "Plantilla_Campo de texto_2" at 638,7 size 59x26; Text 'Fecha:'
   TextField "Plantilla_Campo de texto_3" at 640,39 size 50x26; Text 'Hora:'
   Button "Plantilla_Botón_1" at 464,515 size 80x80; TextOff 'Text'; PictureOff "right-24837_640"
      on Press: ActivateScreen("Cinta chasis", 0)
   Button "Plantilla_Botón_2" at 270,515 size 80x80; TextOff 'Text'; PictureOff "klipartz.com"
      on Press: ActivateScreen("Cinta Rueda", 0)
   Button "Plantilla_Botón_3" at 352,515 size 110x80; TextOff 'Text'; PictureOff "icono casa"
      on Click: ActivateScreen("Control de procesos", 0)
   Button "Plantilla_Botón_4" at 5,515 size 80x80; TextOff 'Text'; PictureOff "seguridad"
      on Press: ActivateScreen("Alarmas", 0)
   Button "Plantilla_Botón_5" at 713,516 size 80x80; TextOff 'Text'; PictureOff "apagar"
      on Click: StopRuntime(0)
   Button "Plantilla_Botón_6" at 89,515 size 80x80; TextOff 'Text'; PictureOff "login"
      on Press: ActivateScreen("Control del usuarios", 0)

screen "Control del usuarios" 800x600, template "Plantilla_1"
   TextField "Campo de texto_1" at 314,105 size 217x26; Text 'CONTROL DE USUARIOS'
      Visibility <- "Es necesario autentificar"
   GraphicView "Visor de gráficos_1" at 499,177 size 172x214; Picture "logout"
   GraphicView "Visor de gráficos_2" at 186,185 size 161x203; Picture "unnamed"
   Button "Botón_1" at 195,397 size 160x32; TextOff 'LOGIN'
      on Press: function_a2a04561()
   Button "Botón_2" at 511,397 size 160x32; TextOff 'LOGOUT'
      on Press: function_f23ef4c9()
   IOField "Campo ES_1" at 222,446 size 400x32; FormatPattern ????????????????????
      ProcessValue <- "Nombre_Usuario"
   TextField "Campo de texto_2" at 233,451 size 152x22; Text 'Sesión iniciada por:'

screen "Cinta Rueda" 800x600, template "Plantilla_1"
   TextField "Campo de texto_5" at 270,77 size 294x37; Text 'CONTROL DE CINTA RUEDAS'
   GraphicView "Visor de gráficos_1" at 42,186 size 734x73; Picture "Screenshot_1"
   GraphicView "Visor de gráficos_5" at 667,139 size 97x47; Picture "Gráfico_7"
   GraphicView "Visor de gráficos_2" at 424,114 size 43x75; Picture "Gráfico_10"
      Visibility <- "Luz cilindro fuera"
   GraphicView "Visor de gráficos_3" at 423,112 size 47x141; Picture "Gráfico_8"
      Visibility <- "Luz cilindro fuera"
   GraphicView "Visor de gráficos_4" at 60,192 size 64x64; Picture "rueda_1"
      Visibility <- "jn cinta lento"
      HorizontalMovement <- "Contador de tiempo"
   GraphicIOField "PlotLight_Round_G_2" at 62,420 size 41x43; PictureOff "PilotLight_Round_G_Off_256c"; PictureOn "PilotLight_Round_G_On_256c"
      ProcessValue <- "Luz cinta rueda"
   GraphicIOField "PlotLight_Round_R_2" at 123,419 size 43x45; PictureOn "PilotLight_Round_R_Off_256c"; PictureOff "PilotLight_Round_R_On_256c"
      ProcessValue <- "Luz cinta rueda"
   Switch "Pushbutton_Round_G_1" at 55,344 size 50x50; CaptionText 'Switch'; TextOff '0'; TextOn '1'; PictureOff "Pushbutton_Round_G_Off_256c"; PictureOn "Pushbutton_Round_G_On_256c"; Authorization "Administración de usuarios"
      on Deactivate: ResetBit("Marcha cinta rueda HMI")
      on Activate: SetBit("Marcha cinta rueda HMI")
      ProcessValue <- "Marcha cinta rueda HMI"
   Switch "Pushbutton_Round_R_1" at 118,344 size 50x50; CaptionText 'Switch'; TextOff '0'; TextOn '1'; PictureOff "Pushbutton_Round_R_Off_256c"; PictureOn "Pushbutton_Round_R_On_256c"; Authorization "Administración de usuarios"
      on Deactivate: ResetBit("Paro cinta rueda HMI")
      on Activate: SetBit("Paro cinta rueda HMI")
      ProcessValue <- "Paro cinta rueda HMI"
   TextField "Campo de texto_9" at 50,318 size 136x22; Text 'MANDO MANUAL'
   TextField "Campo de texto_10" at 52,396 size 118x22; Text 'ESTADO CINTA'
   TextField "Campo de texto_11" at 189,396 size 61x22; Text 'RUEDA'
   GraphicIOField "PlotLight_Round_G_3" at 202,421 size 41x43; PictureOn "PilotLight_Round_G_On_256c"; PictureOff "PilotLight_Round_G_Off_256c"
      ProcessValue <- "Luz rueda en cinta"
   TextField "Campo de texto_12" at 261,396 size 84x22; Text 'CILINDRO'
   GraphicIOField "PlotLight_Round_G_4" at 281,420 size 41x43; PictureOff "PilotLight_Round_G_Off_256c"; PictureOn "PilotLight_Round_G_On_256c"
      ProcessValue <- "Luz cilindro fuera"
   TextField "Campo de texto_13" at 186,318 size 163x22; Text 'CONTROL CILINDRO'
   Switch "Rotary_RG" at 237,339 size 53x55; CaptionText 'Switch'; TextOff '0'; TextOn '1'; PictureOff "Rotary_RG_Off_256c"; PictureOn "Rotary_RG_On_256c"; Authorization "Administración de usuarios"
      on SwitchOff: ResetBit("Control cilindro HMI")
      on SwitchOn: SetBit("Control cilindro HMI")
      ProcessValue <- "Control cilindro HMI"
   Switch "Pushbutton_Emergency" at 634,352 size 102x109; CaptionText 'Switch'; TextOff '0'; TextOn '1'; PictureOff "Pushbutton_Emergency_Off_256c"; PictureOn "Pushbutton_Emergency_On_256c"
      on SwitchOff: ResetBit("Seta emergencia HMI")
      on SwitchOn: SetBit("Seta emergencia HMI")
      ProcessValue <- "Seta emergencia HMI"
   TextField "Campo de texto_1" at 597,322 size 177x22; Text 'PARO DE EMERGENCIA'
   TextField "Campo de texto_2" at 391,322 size 146x22; Text 'VELOCIDAD CINTA'
   Button "Botón_1" at 402,412 size 127x35; TextOff 'AJUSTES'; Authorization "Administración de usuarios"
      on Press: function_efd93a16("Imagen emergente_1", 300, 200, -1, -1, 1)
   IOField "Campo ES_3" at 391,353 size 152x32; FormatPattern 99.9
      ProcessValue <- "Valor frecuencia cinta rueda"
   TextField "Campo de texto_22" at 458,358 size 75x22; Text 'HERCIOS'

screen "Control de procesos" 800x600, template "Plantilla_1"
   Button "Botón_1" at 640,177 size 117x34; TextOff 'MARCHA'; Authorization "Administración de usuarios"
      on Press: SetBit("Marcha HMI")
      on Release: ResetBit("Marcha HMI")
   Button "Botón_2" at 640,231 size 117x34; TextOff 'PARADA'
      on Release: ResetBit("Paro HMI")
      on Press: SetBit("Paro HMI")
   TextField "Campo de texto_1" at 654,119 size 87x22; Text 'MANDO DE'
   TextField "Campo de texto_2" at 654,145 size 80x22; Text 'CONTROL'
   TextField "Campo de texto_3" at 642,321 size 115x22; Text 'INDICADORES'
   TextField "Campo de texto_4" at 647,345 size 104x22; Text 'DE CONTROL'
   GraphicIOField "PlotLight_Round_G" at 642,394 size 50x50; PictureOn "PilotLight_Round_G_On_256c"; PictureOff "PilotLight_Round_G_Off_256c"
      ProcessValue <- "Luz marcha HMI"
   GraphicIOField "PlotLight_Round_R" at 710,394 size 50x50; PictureOn "PilotLight_Round_R_Off_256c"; PictureOff "PilotLight_Round_R_On_256c"
      ProcessValue <- "Luz marcha HMI"
   TextField "Campo de texto_5" at 69,71 size 119x26; Text 'CINTA CHASIS'
   TextField "Campo de texto_6" at 392,71 size 123x26; Text 'CINTA RUEDAS'
   GraphicIOField "PlotLight_Round_G_1" at 62,208 size 50x50; PictureOff "PilotLight_Round_G_Off_256c"; PictureOn "PilotLight_Round_G_On_256c"
      ProcessValue <- "Luz cinta chasis"
   GraphicIOField "PlotLight_Round_R_1" at 126,210 size 50x50; PictureOn "PilotLight_Round_R_Off_256c"; PictureOff "PilotLight_Round_R_On_256c"
      ProcessValue <- "Luz cinta chasis"
   Switch "Pushbutton_Round_G" at 63,132 size 50x50; CaptionText 'Switch'; TextOff '0'; TextOn '1'; PictureOff "Pushbutton_Round_G_Off_256c"; PictureOn "Pushbutton_Round_G_On_256c"; Authorization "Administración de usuarios"
      on Activate: SetBit("Marcha cinta chasis HMI")
      on Deactivate: ResetBit("Marcha cinta chasis HMI")
      ProcessValue <- "Marcha cinta chasis HMI"
   Switch "Pushbutton_Round_R" at 129,132 size 50x50; CaptionText 'Switch'; TextOff '0'; TextOn '1'; PictureOff "Pushbutton_Round_R_Off_256c"; PictureOn "Pushbutton_Round_R_On_256c"; Authorization "Administración de usuarios"
      on Activate: SetBit("Paro cinta chasis HMI")
      on Deactivate: ResetBit("Paro cinta chasis HMI")
      ProcessValue <- "Paro cinta chasis HMI"
   TextField "Campo de texto_7" at 62,110 size 136x22; Text 'MANDO MANUAL'
   TextField "Campo de texto_8" at 43,188 size 165x22; Text 'ESTADO DE LA CINTA'
   GraphicIOField "PlotLight_Round_G_2" at 284,212 size 41x43; PictureOn "PilotLight_Round_G_On_256c"; PictureOff "PilotLight_Round_G_Off_256c"
      ProcessValue <- "Luz cinta rueda"
   GraphicIOField "PlotLight_Round_R_2" at 345,211 size 43x45; PictureOff "PilotLight_Round_R_On_256c"; PictureOn "PilotLight_Round_R_Off_256c"
      ProcessValue <- "Luz cinta rueda"
   Switch "Pushbutton_Round_G_1" at 277,136 size 50x50; CaptionText 'Switch'; TextOff '0'; TextOn '1'; PictureOff "Pushbutton_Round_G_Off_256c"; PictureOn "Pushbutton_Round_G_On_256c"; Authorization "Administración de usuarios"
      on Activate: SetBit("Marcha cinta rueda HMI")
      on Deactivate: ResetBit("Marcha cinta rueda HMI")
      ProcessValue <- "Marcha cinta rueda HMI"
   Switch "Pushbutton_Round_R_1" at 340,136 size 50x50; CaptionText 'Switch'; TextOff '0'; TextOn '1'; PictureOff "Pushbutton_Round_R_Off_256c"; PictureOn "Pushbutton_Round_R_On_256c"; Authorization "Administración de usuarios"
      on Activate: SetBit("Paro cinta rueda HMI")
      on Deactivate: ResetBit("Paro cinta rueda HMI")
      ProcessValue <- "Paro cinta rueda HMI"
   TextField "Campo de texto_9" at 272,110 size 136x22; Text 'MANDO MANUAL'
   TextField "Campo de texto_10" at 274,188 size 118x22; Text 'ESTADO CINTA'
   TextField "Campo de texto_11" at 411,188 size 61x22; Text 'RUEDA'
   GraphicIOField "PlotLight_Round_G_3" at 424,213 size 41x43; PictureOff "PilotLight_Round_G_Off_256c"; PictureOn "PilotLight_Round_G_On_256c"
      ProcessValue <- "Luz rueda en cinta"
   TextField "Campo de texto_12" at 483,188 size 84x22; Text 'CILINDRO'
   GraphicIOField "PlotLight_Round_G_4" at 503,212 size 41x43; PictureOn "PilotLight_Round_G_On_256c"; PictureOff "PilotLight_Round_G_Off_256c"
      ProcessValue <- "Luz cilindro fuera"
   TextField "Campo de texto_13" at 408,110 size 163x22; Text 'CONTROL CILINDRO'
   Switch "Rotary_RG" at 459,131 size 53x55; CaptionText 'Switch'; TextOff '0'; TextOn '1'; PictureOff "Rotary_RG_Off_256c"; PictureOn "Rotary_RG_On_256c"; Authorization "Administración de usuarios"
      on SwitchOn: SetBit("Control cilindro HMI")
      on SwitchOff: ResetBit("Control cilindro HMI")
      ProcessValue <- "Control cilindro HMI"
   Switch "Pushbutton_Emergency" at 55,333 size 133x142; CaptionText 'Switch'; TextOff '0'; TextOn '1'; PictureOff "Pushbutton_Emergency_Off_256c"; PictureOn "Pushbutton_Emergency_On_256c"
      on SwitchOn: SetBit("Seta emergencia HMI")
      on SwitchOff: ResetBit("Seta emergencia HMI")
      ProcessValue <- "Seta emergencia HMI"
   TextField "Campo de texto_14" at 34,286 size 181x26; Text 'PARO DE EMERGENCIA'
   TextField "Campo de texto_15" at 632,71 size 126x26; Text 'MARCHA/PARO'
   TextField "Campo de texto_16" at 264,286 size 311x26; Text 'VARIABLES ANALÓGICAS DEL PROCESO'
   TextField "Campo de texto_17" at 269,324 size 208x22; Text 'VELOCIDAD CINTA CHASIS'
   IOField "Campo ES_1" at 269,346 size 209x32; FormatPattern 99.9
      ProcessValue <- "Velocidades_Velocidad cinta chasis"
   TextField "Campo de texto_18" at 394,351 size 75x22; Text 'HERCIOS'
   TextField "Campo de texto_19" at 268,377 size 281x22; Text 'DISTANCIA CHASIS ULTRASONIDOS'
   IOField "Campo ES_2" at 268,399 size 209x32; FormatPattern 99.99
      ProcessValue <- "Distancia"
   TextField "Campo de texto_20" at 374,404 size 96x22; Text 'Centimetros'
   TextField "Campo de texto_21" at 267,430 size 202x22; Text 'VELOCIDAD CINTA RUEDA'
   IOField "Campo ES_3" at 267,452 size 209x32; FormatPattern 99.9
      ProcessValue <- "Valor frecuencia cinta rueda"
   TextField "Campo de texto_22" at 392,457 size 75x22; Text 'HERCIOS'

screen "Cinta chasis" 800x600, template "Plantilla_1"
   GraphicView "Visor de gráficos_1" at 43,166 size 734x126; Picture "Screenshot_1"
   TextField "Campo de texto_5" at 270,77 size 294x37; Text 'CONTROL DE CINTA CHASIS'
   GraphicView "Visor de gráficos_3" at 16,206 size 36x49; Picture "Gráfico_3"
   GraphicView "Visor de gráficos_4" at 226,172 size 82x112; Picture "pnSDSDSDgwing.com (1)_1"
      HorizontalMovement <- "Ultrasonidos"
   GraphicView "Visor de gráficos_5" at 646,116 size 97x47; Picture "Gráfico_7"
   GraphicIOField "PlotLight_Round_G_1" at 72,422 size 50x50; PictureOn "PilotLight_Round_G_On_256c"; PictureOff "PilotLight_Round_G_Off_256c"
      ProcessValue <- "Luz cinta chasis"
   GraphicIOField "PlotLight_Round_R_1" at 136,424 size 50x50; PictureOff "PilotLight_Round_R_On_256c"; PictureOn "PilotLight_Round_R_Off_256c"
      ProcessValue <- "Luz cinta chasis"
   Switch "Pushbutton_Round_G" at 73,346 size 50x50; CaptionText 'Switch'; TextOff '0'; TextOn '1'; PictureOff "Pushbutton_Round_G_Off_256c"; PictureOn "Pushbutton_Round_G_On_256c"
      on Activate: SetBit("Marcha cinta chasis HMI")
      on Deactivate: ResetBit("Marcha cinta chasis HMI")
      ProcessValue <- "Marcha cinta chasis HMI"
   Switch "Pushbutton_Round_R" at 139,346 size 50x50; CaptionText 'Switch'; TextOff '0'; TextOn '1'; PictureOff "Pushbutton_Round_R_Off_256c"; PictureOn "Pushbutton_Round_R_On_256c"
      on Activate: SetBit("Paro cinta chasis HMI")
      on Deactivate: ResetBit("Paro cinta chasis HMI")
      ProcessValue <- "Paro cinta chasis HMI"
   TextField "Campo de texto_7" at 72,324 size 136x22; Text 'MANDO MANUAL'
   TextField "Campo de texto_8" at 53,402 size 165x22; Text 'ESTADO DE LA CINTA'
   Switch "Pushbutton_Emergency" at 634,355 size 102x109; CaptionText 'Switch'; TextOff '0'; TextOn '1'; PictureOff "Pushbutton_Emergency_Off_256c"; PictureOn "Pushbutton_Emergency_On_256c"
      on SwitchOff: ResetBit("Seta emergencia HMI")
      on SwitchOn: SetBit("Seta emergencia HMI")
      ProcessValue <- "Seta emergencia HMI"
   TextField "Campo de texto_1" at 597,325 size 177x22; Text 'PARO DE EMERGENCIA'
   TextField "Campo de texto_2" at 288,327 size 231x22; Text 'AJUSTE DE VELOCIDAD CINTA'
   IOField "Campo ES_1" at 288,354 size 209x32; Authorization "Administración de usuarios"; FormatPattern 99.9
      ProcessValue <- "Velocidades_Velocidad cinta chasis"
   TextField "Campo de texto_18" at 413,359 size 75x22; Text 'HERCIOS'
   TextField "Campo de texto_19" at 290,401 size 231x22; Text 'DISTANCIA SENSOR - CHASIS'
   IOField "Campo ES_2" at 290,423 size 209x32; FormatPattern 99.99
      ProcessValue <- "Distancia"
   TextField "Campo de texto_20" at 396,428 size 96x22; Text 'Centimetros'

PopupScreen "Imagen emergente_1" 240x240
   TextField "Campo de texto_5" at 18,14 size 152x24; Text 'AJUSTE DE VELOCIDAD'
   Button "Botón_1" at 189,13 size 27x24; TextOff 'X'
      on Press: ActivateScreen("Cinta Rueda", 0)
   TextField "Campo de texto_1" at 24,60 size 150x26; Text 'Velocidad nominal:'
   IOField "Campo ES_1" at 25,90 size 178x32; FormatPattern 99.9
      ProcessValue <- "Velocidades_Velocidad Nominal"
   TextField "Campo de texto_2" at 115,95 size 75x22; Text 'HERCIOS'
   IOField "Campo ES_2" at 28,166 size 178x32; FormatPattern 99.9
      ProcessValue <- "Velocidades_Velocidad Lento"
   TextField "Campo de texto_4" at 115,172 size 75x22; Text 'HERCIOS'
   TextField "Campo de texto_6" at 26,131 size 129x26; Text 'Velocidad lento:'

screen "Alarmas" 800x600, template "Plantilla_1"
   IOField "Campo ES_1" at 387,183 size 166x32; FormatPattern 9999999999999999999999999999999999999999
      ProcessValue <- "Guarda errores_Seta emergencia"
   TextField "Campo de texto_5" at 266,77 size 254x37; Text 'CONTROL DE EMERGENCIAS'
   TextField "Campo de texto_1" at 157,200 size 431x37; Text 'SETA DE EMERGENCIAS:'
   IOField "Campo ES_2" at 394,205 size 186x22; FormatPattern 9999999999999999999999999999999999999999
      ProcessValue <- "Guarda errores_Seta emergencia"
   TextField "Campo de texto_2" at 159,255 size 432x37; Text 'FALLO DETECTA PERSONA:'
   IOField "Campo ES_4" at 395,260 size 186x22; FormatPattern 9999999999999999999999999999999999999999
      ProcessValue <- "Guarda errores_Fallo persona"
   TextField "Campo de texto_3" at 157,312 size 435x37; Text 'FALLO DEL ROBOT:'
   IOField "Campo ES_5" at 394,317 size 186x22; FormatPattern 9999999999999999999999999999999999999999
      ProcessValue <- "Guarda errores_Fallo robot"
   TextField "Campo de texto_4" at 158,368 size 436x37; Text 'GUARDAMOTOR CHASIS:'
   IOField "Campo ES_7" at 393,373 size 186x22; FormatPattern 9999999999999999999999999999999999999999
      ProcessValue <- "Guarda errores_Guardamotor chasis"
   TextField "Campo de texto_6" at 159,424 size 437x37; Text 'GUARDAMOTOR RUEDA:'
   IOField "Campo ES_9" at 394,429 size 186x22; FormatPattern 9999999999999999999999999999999999999999
      ProcessValue <- "Guarda errores_Guardamotor rueda"
   GraphicIOField "PlotLight_Round_R_1" at 608,200 size 37x36; PictureOn "PilotLight_Round_R_On_256c"; PictureOff "PilotLight_Round_R_Off_256c"
      ProcessValue <- "Luz seta emergencia"
   GraphicIOField "PlotLight_Round_R_2" at 609,255 size 37x36; PictureOff "PilotLight_Round_R_Off_256c"; PictureOn "PilotLight_Round_R_On_256c"
      ProcessValue <- "Luz fallo persona"
   GraphicIOField "PlotLight_Round_R_3" at 609,313 size 37x36; PictureOff "PilotLight_Round_R_Off_256c"; PictureOn "PilotLight_Round_R_On_256c"
      ProcessValue <- "Luz fallo robot"
   GraphicIOField "PlotLight_Round_R_4" at 608,368 size 37x36; PictureOff "PilotLight_Round_R_Off_256c"; PictureOn "PilotLight_Round_R_On_256c"
      ProcessValue <- "Luz guardamotor chasis"
   GraphicIOField "PlotLight_Round_R_5" at 609,426 size 37x36; PictureOff "PilotLight_Round_R_Off_256c"; PictureOn "PilotLight_Round_R_On_256c"
      ProcessValue <- "Luz guardamotor rueda"
   TextField "Campo de texto_7" at 249,152 size 297x22; Text 'REGISTRO DE ÚLTIMAS EMERGENCIAS'

scheduled task "Leer nombre de usuario"
   on Action: function_f41c6f6c("Nombre_Usuario"); ActivateScreen("Control de procesos", 0)
*)